FUNCTION_BLOCK FB79
TITLE = 'process_F1'
AUTHOR : CB

VAR
	tmp : BOOL;
END_VAR


BEGIN


NETWORK
TITLE =
//
//	process/process_F1/FloMGT1PROC
CALL FC78 (combE := 1);
CALL FB78,	DB78;
CALL FC78 (combE := 0);




END_FUNCTION_BLOCK
